// TwinCAT 3 PLC project PRG_HMIElements
// Title: B_HMIElements
// Company: RafalOS
// Author: Rafał Osajda
// ProjectVersion: 0.0.0.7
// ProgramVersion: 3.1.4024.0
// libraries:
//   B_Base, * (RafalOS)
//   B_Base_HMI_Connector, * (RafalOS)
//   Tc2_Standard, * (Beckhoff Automation GmbH)
//   Tc2_System, * (Beckhoff Automation GmbH)
//   Tc3_Module, * (Beckhoff Automation GmbH)
// project tree:
//   GVLs/ GVL_HMIEConstans.TcGVL
//   / PlcTask.TcTTO (not stored)
//   POUs Compilation/ PRG_Compilation.TcPOU
//   POUs/01A_Button/ FB_HMIEButton.TcPOU (not stored), ITF_HMIEButton.TcIO, ITF_HMIEButton_HMI_Connector.TcIO, ITF_HMIEButton_HMI_Init.TcIO
//   POUs/01B_ButtonHMI/ FB_HMIEButton_HMI.TcPOU, ITF_HMIEButton_HMI.TcIO, ST_HMIEButton_HMI.TcDUT, ST_HMIEButton_HMI_Link.TcDUT (not stored)
//   POUs/02A_Menu/ FB_HMIEMenu.TcPOU, ITF_HMIEMenu_HMI_Connector.TcIO (not stored), ITF_HMIEMenu_HMI_Init.TcIO (not stored), ITF_HMIEMenu.TcIO
//   POUs/02B_MenuHMI/ FB_HMIEMenu_HMI.TcPOU, ITF_HMIEMenu_HMI.TcIO, ST_HMIEMenu_HMI.TcDUT, ST_HMIEMenu_HMI_Link.TcDUT
// real-time tasks:
//   TASK PlcTask: cycle T#10ms, priority 20, ADS port 350

// ---- POUs/01B_ButtonHMI/ST_HMIEButton_HMI.TcDUT
TYPE ST_HMIEButton_HMI :
STRUCT
	bActive		: BOOL;
	bVisible	: BOOL;
	bEnable		: BOOL;
	bPushed		: BOOL;
END_STRUCT
END_TYPE

// ---- POUs/02B_MenuHMI/ST_HMIEMenu_HMI.TcDUT
TYPE ST_HMIEMenu_HMI :
STRUCT
	iNumberOfActivePage			: INT;
	iNumberOfAddedScreen		: INT;
	wsTitleActivePage			: WSTRING;
	bChangePage					: BOOL;
END_STRUCT
END_TYPE

// ---- POUs/02B_MenuHMI/ST_HMIEMenu_HMI_Link.TcDUT
TYPE ST_HMIEMenu_HMI_Link EXTENDS ST_BaseControlElement_HMI_Link :
STRUCT
	stMenu					: ST_HMIEMenu_HMI;
	arrButton				: ARRAY [0..GVL_HMIEConstans.MAX_NUMBER_OF_BUTTON_IN_MENU] OF ST_HMIEButton_HMI_Link;
END_STRUCT
END_TYPE

// ---- GVLs/GVL_HMIEConstans.TcGVL
{attribute 'qualified_only'}
VAR_GLOBAL CONSTANT
	MAX_NUMBER_OF_BUTTON_IN_MENU	: INT := 20;
	
END_VAR

// ---- POUs/01A_Button/ITF_HMIEButton.TcIO
INTERFACE ITF_HMIEButton EXTENDS ITF_BaseComponent

METHOD PUBLIC IsActive : BOOL
VAR_INPUT
END_VAR
END_METHOD

METHOD PUBLIC IsEnable : BOOL
VAR_INPUT
END_VAR
END_METHOD

METHOD PUBLIC IsPressed : BOOL
VAR_INPUT
END_VAR
END_METHOD

METHOD PUBLIC IsVisible : BOOL
VAR_INPUT
END_VAR
END_METHOD

METHOD PUBLIC SetActive
VAR_INPUT
	bIN: BOOL;
END_VAR
END_METHOD

METHOD PUBLIC SetEnable
VAR_INPUT
	bIN: BOOL;
END_VAR
END_METHOD

METHOD PUBLIC SetPressed
VAR_INPUT
	bIN: BOOL;
END_VAR
END_METHOD

METHOD PUBLIC SetVisible
VAR_INPUT
	bIN: BOOL;
END_VAR
END_METHOD

END_INTERFACE

// ---- POUs/01A_Button/ITF_HMIEButton_HMI_Connector.TcIO
(*			
	RafalOS
	Rafał Osajda		12.11.2025		TC 4024.66
	Zbiór metod umożliwiające odczyt danych z hmi 
*)
INTERFACE ITF_HMIEButton_HMI_Connector EXTENDS ITF_BaseComponent_HMI_Connector

METHOD PUBLIC IsActive : BOOL
VAR_INPUT
END_VAR
END_METHOD

METHOD PUBLIC IsEnable : BOOL
VAR_INPUT
END_VAR
END_METHOD

METHOD PUBLIC IsPressed : BOOL
VAR_INPUT
END_VAR
END_METHOD

METHOD PUBLIC IsVisible : BOOL
VAR_INPUT
END_VAR
END_METHOD

METHOD PUBLIC SetPressed
VAR_INPUT
	bIN: BOOL;
END_VAR
END_METHOD

END_INTERFACE

// ---- POUs/01A_Button/ITF_HMIEButton_HMI_Init.TcIO
(*			
	RafalOS
	Rafał Osajda		12.11.2025		TC 4024.66
	interfejs do przekazywania przy tworzeniu elementów
*)
INTERFACE ITF_HMIEButton_HMI_Init EXTENDS ITF_BaseComponent, ITF_HMIEButton_HMI_Connector

END_INTERFACE

// ---- POUs/01B_ButtonHMI/ITF_HMIEButton_HMI.TcIO
(*			
	RafalOS
	Rafał Osajda		12.11.2025		TC 4024.66
	interfejs potrzebny w HMI
*)
INTERFACE ITF_HMIEButton_HMI EXTENDS ITF_BaseComponent_HMI

METHOD PUBLIC GetNameOfButton : WSTRING
VAR_INPUT
END_VAR
END_METHOD

METHOD LinkHMIEButtonData : BOOL
VAR_INPUT
	stData					: REFERENCE TO ST_HMIEButton_HMI_Link;
END_VAR
END_METHOD

END_INTERFACE

// ---- POUs/02A_Menu/ITF_HMIEMenu.TcIO
INTERFACE ITF_HMIEMenu EXTENDS ITF_BaseControlElement

METHOD PUBLIC GetNumberOfActriveScreen : INT
VAR_INPUT
END_VAR
END_METHOD

METHOD PUBLIC GetNumberOfAddedButton : INT
VAR_INPUT
END_VAR
END_METHOD

METHOD IsActiveButton : BOOL
VAR_INPUT
	iButton		: INT;	//numer przycisku
	bIN			: BOOL;
END_VAR
END_METHOD

METHOD PUBLIC IsChangePage : BOOL
VAR_INPUT
END_VAR
END_METHOD

METHOD IsEnableButton : BOOL
VAR_INPUT
	iButton		: INT;	//numer przycisku
	bIN			: BOOL;
END_VAR
END_METHOD

METHOD IsVisibleButton : BOOL
VAR_INPUT
	iButton		: INT;	//numer przycisku
	bIN			: BOOL;
END_VAR
END_METHOD

METHOD PUBLIC ResetChangePage
VAR_INPUT
END_VAR
END_METHOD

METHOD SetActiveButton : BOOL
VAR_INPUT
	iButton		: INT;	//numer przycisku
	bIN			: BOOL;
END_VAR
END_METHOD

METHOD SetEnableButton : BOOL
VAR_INPUT
	iButton		: INT;	//numer przycisku
	bIN			: BOOL;
END_VAR
END_METHOD

METHOD SetVisibleButton : BOOL
VAR_INPUT
	iButton		: INT;	//numer przycisku
	bIN			: BOOL;
END_VAR
END_METHOD

(*			
	RafalOS
	Rafał Osajda		11.11.2025		TC 4024.66
	testuje czy jest coś naciśnięte w menu i przełącza
*)
METHOD PUBLIC Testing : BOOL
END_METHOD

END_INTERFACE

// ---- POUs/02B_MenuHMI/ITF_HMIEMenu_HMI.TcIO
(*			
	RafalOS
	Rafał Osajda		12.11.2025		TC 4024.66
	interfejs potrzebny w HMI
*)
INTERFACE ITF_HMIEMenu_HMI EXTENDS ITF_BaseControlElement_HMI

(*			
	RafalOS
	Rafał Osajda		18.11.2025		TC 4024.66
	Pobiera numer aktywnej strony menu głównego
*)
METHOD GetNumberOfActiveScreen : INT
VAR_INPUT
END_VAR
END_METHOD

(*			
	RafalOS
	Rafał Osajda		18.11.2025		TC 4024.66
	Pobiera numer aktywnej strony menu głównego
*)
METHOD GetNumberOfPreviewScreen : INT
VAR_INPUT
END_VAR
END_METHOD

(*			
	RafalOS
	Rafał Osajda		18.11.2025		TC 4024.66
	Pobiera tytuł z aktywnej strony
*)
METHOD GetTitleOfActualScreen : WSTRING
VAR_INPUT
END_VAR
END_METHOD

METHOD PUBLIC IsChangePage : BOOL
VAR_INPUT
END_VAR
END_METHOD

METHOD LinkHMIEMenuData : BOOL
VAR_INPUT
	stData				: reference to ST_HMIEMenu_HMI_Link;
END_VAR
END_METHOD

END_INTERFACE

// ---- POUs Compilation/PRG_Compilation.TcPOU
PROGRAM PRG_Compilation
VAR
	fbLogger		: FB_BaseLogger;
	fbButton		: FB_HMIEButton;
	fbButtonHMI		: FB_HMIEButton_HMI (itfBaseLoggerConnector := fbLogger, itfButton := fbButton);
	fbMenu			: FB_HMIEMenu;
	fbMenuHMI		: FB_HMIEMenu_HMI (itfBaseLoggerConnector := fbLogger, itfMenu := fbMenu);
END_VAR

END_PROGRAM

// ---- POUs/01B_ButtonHMI/FB_HMIEButton_HMI.TcPOU
FUNCTION_BLOCK FB_HMIEButton_HMI EXTENDS FB_BaseComponent_HMI IMPLEMENTS ITF_HMIEButton_HMI
VAR
	itfButton			: ITF_HMIEButton_HMI_Connector;
	refstButtonData		: REFERENCE TO ST_HMIEButton_HMI;
END_VAR

METHOD FB_init : BOOL
VAR_INPUT
	bInitRetains 	: BOOL; // if TRUE, the retain variables are initialized (warm start / cold start)
	bInCopyCode 	: BOOL;  // if TRUE, the instance afterwards gets moved into the copy code (online change)
	itfBaseLoggerConnector	: ITF_BaseLogger_HMI_Connector;	//bezpośredni łącznik do logera
	itfButton				: ITF_HMIEButton_HMI_Init;
END_VAR
THIS^.itfButton := itfButton;
//Przypisanie do elementów z biblioteki
THIS^.itfBaseLoggerElementConnector := itfbutton;
THIS^.itfBaseComponentConnector := itfbutton;

//
THIS^.itfBaseLoggerConnector := itfBaseLoggerConnector;

IF (THIS^.itfButton <> 0 AND
	THIS^.itfBaseLoggerElementConnector <> 0 AND
	THIS^.itfBaseComponentConnector	<> 0 AND
	THIS^.itfBaseLoggerConnector <> 0) THEN
	THIS^.bIsInit						:= TRUE;
END_IF
END_METHOD

METHOD PUBLIC GetNameOfButton : WSTRING
VAR_INPUT
END_VAR
GetNameOfButton := GetTextFromLabelForActiveLocation (stLabel := this^.itfButton.GetName ());
END_METHOD

METHOD LinkHMIEButtonData : BOOL
VAR_INPUT
	stData					: REFERENCE TO ST_HMIEButton_HMI_Link;
END_VAR
THIS^.refstButtonData REF= stData.stButtonHMI;

THIS^.refstBaseLoggerElementDataHMI REF= stData.stBaseLoggerElement;
THIS^.refstBaseComponentDataHMI REF= stData.stBaseComponent;

THIS^.CreateLinkToEventsMemory ();

IF (__ISVALIDREF (THIS^.refstButtonData) AND THIS^.IsLinkedReferences ()) THEN
	THIS^.bIsValidData := TRUE;
	LinkHMIEButtonData := TRUE;
END_IF
END_METHOD

(*			
	RafalOS
	Rafał Osajda		14.11.2025		TC 4024.66
	Metoda przygotowywania danych dla HMI 
	W niej odbywa się odpytywanie właściego elementu przez łącznik
*)
METHOD PUBLIC PrepareDataForHMI : BOOL
VAR_INPUT
END_VAR
SUPER^.PrepareDataForHMI ();

IF (THIS^.refstButtonData.bPushed) THEN
	THIS^.refstButtonData.bPushed := FALSE;
	THIS^.itfButton.SetPressed (bIN := TRUE);
END_IF

THIS^.refstButtonData.bActive := THIS^.itfButton.IsActive ();
THIS^.refstButtonData.bEnable := THIS^.itfButton.IsEnable ();
THIS^.refstButtonData.bVisible := THIS^.itfButton.IsVisible ();
END_METHOD

END_FUNCTION_BLOCK

// ---- POUs/02A_Menu/FB_HMIEMenu.TcPOU
FUNCTION_BLOCK FB_HMIEMenu EXTENDS FB_BaseControlElement IMPLEMENTS ITF_HMIEMenu, ITF_HMIEMenu_HMI_Init
VAR
	arrButtons				: ARRAY [0..GVL_HMIEConstans.MAX_NUMBER_OF_BUTTON_IN_MENU] OF ITF_HMIEButton;
	iNumberOfButton			: INT := -1;	//ilosć przycisków w menu
	iActiveButton			: INT;	//numer aktywnego przycisku
	iActiveButtonPrev		: INT;
	bChangePage				: BOOL; //zmiana strony
END_VAR

METHOD PUBLIC AddButton : BOOL
VAR_INPUT
	fbButton			: ITF_HMIEButton;
END_VAR
IF (THIS^.iNumberOfButton + 1 <= GVL_HMIEConstans.MAX_NUMBER_OF_BUTTON_IN_MENU) THEN
	THIS^.iNumberOfButton := THIS^.iNumberOfButton + 1;
	THIS^.arrButtons [THIS^.iNumberOfButton] := fbButton;
	THIS^.arrButtons [THIS^.iNumberOfButton].SetEnable (bIN := TRUE);
	THIS^.arrButtons [THIS^.iNumberOfButton].SetVisible (bIN := TRUE);
	THIS^.AddComponent (itfComponent := fbButton);
	AddButton := TRUE;
ELSE
	AddButton := FALSE;
END_IF
END_METHOD

METHOD PUBLIC GetNumberOfActrivePreviewScreen : INT
VAR_INPUT
END_VAR
GetNumberOfActrivePreviewScreen := THIS^.iActiveButtonPrev;
END_METHOD

METHOD PUBLIC GetNumberOfActriveScreen : INT
VAR_INPUT
END_VAR
GetNumberOfActriveScreen := THIS^.iActiveButton;
END_METHOD

METHOD PUBLIC GetNumberOfAddedButton : INT
VAR_INPUT
END_VAR
GetNumberOfAddedButton := THIS^.iNumberOfButton;
END_METHOD

METHOD PUBLIC GetTitleOfActivePage : WSTRING
VAR_INPUT
END_VAR
//GetTitleOfActivePage := this^.arrButtons [this^.iActiveButton].GetName ();
END_METHOD

METHOD IsActiveButton : BOOL
VAR_INPUT
	iButton		: INT;	//numer przycisku
	bIN			: BOOL;
END_VAR
IsActiveButton	:= THIS^.arrButtons [iButton].IsActive ();
END_METHOD

METHOD PUBLIC IsChangePage : BOOL
VAR_INPUT
END_VAR
IsChangePage := THIS^.bChangePage;
END_METHOD

METHOD IsEnableButton : BOOL
VAR_INPUT
	iButton		: INT;	//numer przycisku
	bIN			: BOOL;
END_VAR
IsEnableButton	:= THIS^.arrButtons [iButton].IsEnable ();
END_METHOD

METHOD IsVisibleButton : BOOL
VAR_INPUT
	iButton		: INT;	//numer przycisku
	bIN			: BOOL;
END_VAR
IsVisibleButton	:= THIS^.arrButtons [iButton].IsVisible ();
END_METHOD

METHOD PUBLIC ResetChangePage
VAR_INPUT
END_VAR
THIS^.bChangePage := FALSE;
END_METHOD

METHOD SetActiveButton : BOOL
VAR_INPUT
	iButton		: INT;	//numer przycisku
	bIN			: BOOL;
END_VAR
THIS^.arrButtons [iButton].SetActive (bIN := bIN);
END_METHOD

METHOD SetEnableButton : BOOL
VAR_INPUT
	iButton		: INT;	//numer przycisku
	bIN			: BOOL;
END_VAR
THIS^.arrButtons [iButton].SetEnable (bIN := bIN);
END_METHOD

METHOD SetVisibleButton : BOOL
VAR_INPUT
	iButton		: INT;	//numer przycisku
	bIN			: BOOL;
END_VAR
THIS^.arrButtons [iButton].SetVisible (bIN := bIN);
END_METHOD

(*			
	RafalOS
	Rafał Osajda		11.11.2025		TC 4024.66
	testuje czy jest coś naciśnięte w menu i przełącza
*)
METHOD PUBLIC Testing : BOOL
VAR
	iI		: INT;
	iJ		: INT;
END_VAR
FOR iI := 0 TO THIS^.iNumberOfButton DO
	IF (THIS^.arrButtons [iI].IsPressed ()) THEN
		FOR iJ := 0 TO THIS^.iNumberOfButton DO 
			THIS^.arrButtons [iJ].SetActive (bIN := FALSE);
		END_FOR
		THIS^.arrButtons [iI].SetPressed (bIN := FALSE);
		THIS^.arrButtons [iI].SetActive (bIN := TRUE);
		THIS^.iActiveButtonPrev := THIS^.iActiveButton;
		THIS^.iActiveButton := iI;
		THIS^.bChangePage := TRUE;
	END_IF
END_FOR
END_METHOD

END_FUNCTION_BLOCK

// ---- POUs/02B_MenuHMI/FB_HMIEMenu_HMI.TcPOU
FUNCTION_BLOCK FB_HMIEMenu_HMI EXTENDS FB_BaseControlElement_HMI IMPLEMENTS ITF_HMIEMenu_HMI
VAR
	itfMenu			: ITF_HMIEMenu_HMI_Connector;
	refstMenuData	: REFERENCE TO ST_HMIEMenu_HMI;

	arrButtons		: ARRAY [0..GVL_HMIEConstans.MAX_NUMBER_OF_BUTTON_IN_MENU] OF ITF_HMIEButton_HMI;
	
END_VAR

METHOD PUBLIC AddButton : BOOL
VAR_INPUT
	fbButtonHMI			: ITF_HMIEButton_HMI;
END_VAR
THIS^.AddComponent (itfComponentHMI := fbButtonHMI);
THIS^.arrButtons [THIS^.uiNumberOfComponents - 1] := fbButtonHMI;
END_METHOD

METHOD FB_init : BOOL
VAR_INPUT
	bInitRetains : BOOL; // if TRUE, the retain variables are initialized (warm start / cold start)
	bInCopyCode : BOOL;  // if TRUE, the instance afterwards gets moved into the copy code (online change)
	itfBaseLoggerConnector	: ITF_BaseLogger_HMI_Connector;	//bezpośredni łącznik do logera
	itfMenu			: ITF_HMIEMenu_HMI_Init;
END_VAR
THIS^.itfMenu := itfMenu;

//Przypisanie do elementów z biblioteki
THIS^.itfBaseLoggerElementConnector		:= itfMenu;
THIS^.itfBaseComponentConnector			:= itfMenu;
THIS^.itfBaseControlElementConnector	:= itfMenu;
//
THIS^.itfBaseLoggerConnector			:= itfBaseLoggerConnector;
//

IF (THIS^.itfMenu <> 0 AND
	THIS^.itfBaseLoggerElementConnector <> 0 AND
	THIS^.itfBaseComponentConnector	<> 0 AND
	THIS^.itfBaseControlElementConnector <> 0 AND
	THIS^.itfBaseLoggerConnector <> 0) THEN
	THIS^.bIsInit						:= TRUE;
END_IF
END_METHOD

(*			
	RafalOS
	Rafał Osajda		18.11.2025		TC 4024.66
	Pobiera numer aktywnej strony menu głównego
*)
METHOD GetNumberOfActiveScreen : INT
VAR_INPUT
END_VAR
GetNumberOfActiveScreen := THIS^.itfMenu.GetNumberOfActriveScreen ();
END_METHOD

(*			
	RafalOS
	Rafał Osajda		18.11.2025		TC 4024.66
	Pobiera numer aktywnej strony menu głównego
*)
METHOD GetNumberOfPreviewScreen : INT
VAR_INPUT
END_VAR
GetNumberOfPreviewScreen := THIS^.itfMenu.GetNumberOfActrivePreviewScreen ();
END_METHOD

(*			
	RafalOS
	Rafał Osajda		18.11.2025		TC 4024.66
	Pobiera tytuł z aktywnej strony
*)
METHOD GetTitleOfActualScreen : WSTRING
VAR_INPUT
END_VAR
GetTitleOfActualScreen := THIS^.GetTextFromLabelForActiveLocation (stLabel := THIS^.itfMenu.GetName ());
END_METHOD

METHOD PUBLIC IsChangePage : BOOL
VAR_INPUT
END_VAR
IsChangePage := THIS^.itfMenu.IsChangePage ();
END_METHOD

METHOD LinkHMIEMenuData : BOOL
VAR_INPUT
	stData				: reference to ST_HMIEMenu_HMI_Link;
END_VAR
VAR
	iI					: INT;
END_VAR
THIS^.refstMenuData REF= stData.stMenu;	//ta zmienna powstaje w elemencie 

THIS^.refstBaseLoggerElementDataHMI REF= stData.stBaseLoggerElement;	//zmienne z biblioteki ale dopiero tu je moge przypisać 
THIS^.refstBaseComponentDataHMI REF= stData.stBaseComponent;
THIS^.refstBaseControlElementDataHMI REF= stData.stBaseControlElement;

FOR iI := 0 TO GVL_HMIEConstans.MAX_NUMBER_OF_BUTTON_IN_MENU DO
	IF (THIS^.arrButtons [iI] <> 0) THEN
		THIS^.arrButtons [iI].LinkHMIEButtonData (stData := stData.arrButton [iI]);
	END_IF
END_FOR


THIS^.CreateLinkToEventsMemory ();	//wywołanie metody linkującą poamięc zgłoszęń

IF (__ISVALIDREF (THIS^.refstMenuData) AND THIS^.IsLinkedReferences ()) THEN
	THIS^.bIsValidData := TRUE;
	LinkHMIEMenuData := TRUE;
END_IF
END_METHOD

(*			
	RafalOS
	Rafał Osajda		14.11.2025		TC 4024.66
	Metoda przygotowywania danych dla HMI 
	W niej odbywa się odpytywanie właściego elementu przez łącznik
*)
METHOD PUBLIC PrepareDataForHMI : BOOL
VAR_INPUT
END_VAR

VAR
	iI: INT;
END_VAR
SUPER^.PrepareDataForHMI ();

THIS^.refstMenuData.iNUmberOfActivePage := THIS^.itfMenu.GetNumberOfActriveScreen ();
THIS^.refstMenuData.iNumberOfAddedScreen := THIS^.itfMenu.GetNumberOfAddedButton ();

FOR iI := 0 TO THIS^.refstMenuData.iNumberOfAddedScreen  DO
	THIS^.arrButtons [iI].PrepareDataForHMI ();
END_FOR


THIS^.refstMenuData.wsTitleActivePage := THIS^.arrButtons [THIS^.refstMenuData.iNUmberOfActivePage].GetNameOfButton ();
THIS^.refstMenuData.bChangePage := THIS^.itfMenu.IsChangePage ();
END_METHOD

END_FUNCTION_BLOCK
